{attribute 'linkalways'} 
{attribute 'no_explicit_call' := 'This FB is a CLASS and must be accessed using methods or properties'}
{attribute 'enable_dynamic_creation'}
FUNCTION_BLOCK _LREAL EXTENDS NumericDatatypeBase
VAR
	localData : LREAL;
	activeData : REFERENCE TO LREAL REF= localData;
END_VAR

PROPERTY PUBLIC Address : PVOID
GET
Address := ADR(activeData);
END_GET
END_PROPERTY

METHOD PUBLIC ClearReference
VAR_INPUT
END_VAR
activeData REF= localData;
END_METHOD

METHOD PUBLIC Clone : I_Datatype
VAR
    pClone : POINTER TO _LREAL;
END_VAR
pClone := __NEW(_LREAL(InitialValue := Value));
Clone := pClone^;
END_METHOD

METHOD FB_init : BOOL
VAR_INPUT
	bInitRetains : BOOL; // if TRUE, the retain variables are initialized (warm start / cold start)
	bInCopyCode : BOOL;  // if TRUE, the instance afterwards gets moved into the copy code (online change)
	InitialValue : LREAL;
END_VAR
localData := InitialValue;
END_METHOD

PROPERTY PUBLIC IsFloat : BOOL
GET
IsFloat := TRUE;
END_GET
END_PROPERTY

PROPERTY PUBLIC IsSigned : BOOL
GET
IsSigned := TRUE;
END_GET
END_PROPERTY

METHOD PUBLIC MakeReferenceTo
VAR_INPUT
	ReferenceTarget : REFERENCE TO LREAL;
END_VAR
activeData REF= ReferenceTarget;
END_METHOD

PROPERTY PUBLIC MaxValue : LREAL
GET
MaxValue :=  DatatypeLimits.LREAL_MAX_VALUE;
END_GET
END_PROPERTY

PROPERTY PUBLIC MinValue : LREAL
GET
MinValue := DatatypeLimits.LREAL_MIN_VALUE;
END_GET
END_PROPERTY

METHOD PROTECTED SerializeMaxValue
VAR_INPUT
	Serializer : I_Serializer;
END_VAR
Serializer.AddLreal(MaxValue);
END_METHOD

METHOD PROTECTED SerializeMinValue
VAR_INPUT
	Serializer : I_Serializer;
END_VAR
Serializer.AddLreal(MinValue);
END_METHOD

METHOD PUBLIC SerializeWith
VAR_INPUT
	Serializer : I_Serializer;
END_VAR
Serializer.AddLreal(activeData);
END_METHOD

PROPERTY PUBLIC Size : UDINT
GET
Size := SIZEOF(activeData);
END_GET
END_PROPERTY

METHOD TryDeserializeFrom : BOOL
VAR_INPUT
	Deserializer : I_Deserializer;
	Feedback : I_DeserializerFeedback;
END_VAR
TryDeserializeFrom := Deserializer.TryGetLreal(activeData, Feedback);
END_METHOD

METHOD TryMakeReferenceTo : BOOL
VAR_INPUT
	Target : I_Datatype;
END_VAR
VAR
	pTargetData : POINTER TO LREAL;
END_VAR
IF NOT (Target.TypeName = TypeName) THEN
	RETURN;
END_IF

pTargetData := Target.Address;
activeData REF= pTargetData^;
TryMakeReferenceTo := TRUE;
END_METHOD

PROPERTY PUBLIC TypeName : T_MAXSTRING
GET
TypeName := 'LREAL';
END_GET
END_PROPERTY

PROPERTY PUBLIC Value : REFERENCE TO LREAL
GET
Value REF= activeData;
END_GET
END_PROPERTY

END_FUNCTION_BLOCK

(* stored: Version 1.1.0.1, ProductVersion 3.1.4024.12
   POU _LREAL: Id {cc05ec20-dde3-4620-8951-148abfb0053c}, SpecialFunc None
   Folder Constructor: Id {a934c424-137d-42f8-af4c-56343d1f2818}
   Folder Protected: Id {7e4d9fa1-9695-0f1c-1c1e-6915e9123158}
   Property Address: Id {cc0072cc-c616-423d-842c-0b4a616cde59}
   Get Get: Id {f49a81b8-f747-47ee-b8dd-73af7e334361}
   Method ClearReference: Id {843a3718-36d8-45a2-b963-ae06c440e19b}
   Method Clone: Id {f58a1f4f-5066-4158-9eca-2c67cf283a3a}
   Method FB_init: Id {f1ccfb84-1244-45ac-8c76-9fcb512a9f94}
   Property IsFloat: Id {ced1409c-3953-48b6-ab91-a12814ed569b}
   Get Get: Id {f608de6f-3bad-49d8-b002-970549314be5}
   Property IsSigned: Id {ecee7cea-9782-4cd9-bf0d-b432c5958e0b}
   Get Get: Id {8c971876-b10e-488c-9e2a-56c35c9b1a1b}
   Method MakeReferenceTo: Id {cdd8d06f-e9fd-4897-b1a5-1b9b17752db1}
   Property MaxValue: Id {8cbb32e8-4299-07d9-0fed-f377845df685}
   Get Get: Id {8bfd8fc2-64b9-0b1f-39a5-a998a0ac598a}
   Property MinValue: Id {74151111-62ab-09d5-27cd-23a52b8a6797}
   Get Get: Id {d7968ca9-5a4d-0ba5-02bd-083a644a05d6}
   Method SerializeMaxValue: Id {45955609-ed01-05c3-2d38-ae2d5ec2865d}
   Method SerializeMinValue: Id {650de54f-321c-0504-3ebc-55346f957ca0}
   Method SerializeWith: Id {02aabc19-6942-48ee-8f2d-313a86b52ff9}
   Property Size: Id {89c261d1-bac6-4392-bda7-50836f50db6e}
   Get Get: Id {5a1892e8-9d04-4dbd-a8fb-385510d4753c}
   Method TryDeserializeFrom: Id {331ced44-7540-4591-a72e-5e6d03d318cc}
   Method TryMakeReferenceTo: Id {ee5954bf-2a0d-483b-8886-91a0bb74a20d}
   Property TypeName: Id {a432f784-e285-4645-9d2e-b5735c558c9d}
   Get Get: Id {fa4e0604-e362-454f-bf9c-31636f2adae8}
   Property Value: Id {27002f84-6748-4a80-8b6e-791fe85a74b0}
   Get Get: Id {d571196e-195c-458a-90d9-7091d9058e54} *)
